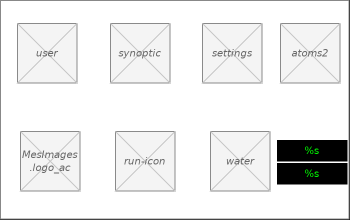
VISUALIZATION VISU_BANDEAU  // 350x220
VAR_INPUT
	m_Input_MACHINE : BLOCK_MODE_MARCHE_V2_0;
END_VAR
    Rectangle (0,0 350x220)
    Image (115,131 60x60), image: run-icon
        toggle Global_Variables.SHOW_SM_SA
        OnMouseClick: change screen: VISU_SA
    Image (202,23 60x60), image: settings
        OnMouseClick: execute { Global_Variables.SHOW_SM_SA:=(FALSE); }
        OnMouseClick: change screen: VISU_CONFIG_POMPAGE
    Image (17,23 60x60), image: user
        OnMouseClick: execute { Global_Variables.SHOW_SM_SA:=(FALSE); }
        OnMouseClick: change screen: UTIL_MENU
    Image (20,131 60x60), image: MesImages.logo_ac
        OnMouseClick: execute { Global_Variables.SHOW_SM_SA:=(FALSE); }
        OnMouseClick: change screen: SYN_INFOS
    Image (110,23 60x60), image: synoptic
        OnMouseClick: execute { Global_Variables.SHOW_SM_SA:=(FALSE); }
        OnMouseClick: change screen: SYN_PROC
    Image (210,131 60x60), image: water
        OnMouseClick: execute { Global_Variables.SHOW_SM_SA:=(FALSE); }
        OnMouseClick: change screen: SYN_SERVITUDES
    Image (280,23 60x60), image: atoms2
        OnMouseClick: execute { Global_Variables.SHOW_SM_SA:=(FALSE); }
        OnMouseClick: change screen: SYN_EXEC_PROC
    Rectangle (277,163 70x21), "%s", text variable: PRG_SEC.STATE_Time
    Rectangle (277,140 70x21), "%s", text variable: PRG_SEC.STATE_Date
END_VISUALIZATION

(* stored: Version 1.1.0.1, ProductVersion 3.1.4024.12
   Visu VISU_BANDEAU: Id {0f1ed10f-d5e3-499d-b683-8f98a266eec9} *)
